FUNCTION_BLOCK FB_Manual_Mode
VAR_INPUT
    Number_Of_Switches      : USINT;
    Switch_Status           : ARRAY[1..8] OF BOOL;
    Switch_Power            : ARRAY[1..8] OF REAL;
END_VAR
VAR_OUTPUT
    Target_Power_kW         : REAL;
END_VAR
VAR
    i                       : USINT;
END_VAR

Target_Power_kW := 0.0;

FOR i := 1 TO Number_Of_Switches DO
    IF Switch_Status[i] THEN
        Target_Power_kW := Target_Power_kW + Switch_Power[i];
    END_IF;
END_FOR;

END_FUNCTION_BLOCK

(* stored: Version 1.1.0.1, ProductVersion 3.1.4024.16
   POU FB_Manual_Mode: Id {dccf7914-1417-4283-ac53-e4dbde30632b}, SpecialFunc None *)
